FUNCTION_BLOCK SludgeBufferLogic_2 (* Composite Function Block Type *)
  (* Standard: 61499-2 *)
  (* Version 1.3, 10/1/2026, Claude/Hidryco, Schneider Electric, Rev1.3 - Revertidas as ligacoes de emergencia da Rev1.2 (FB_* e comando nos Av) que fechavam laco de eventos com a receita de emergencia; igual a Rev1.1 *)
  PACKAGE SE.Nereda;
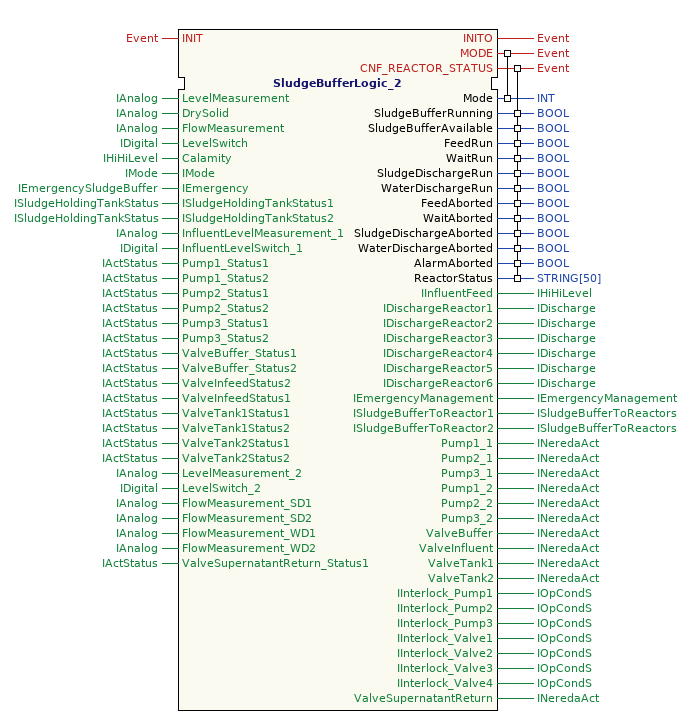
  EVENT_INPUT
    INIT; (* Initialization Request *)
  END_EVENT
  EVENT_OUTPUT
    INITO; (* Initialization Confirm *)
    MODE WITH Mode; (* Response from Socket *)
    CNF_REACTOR_STATUS WITH SludgeBufferRunning, SludgeBufferAvailable, FeedAborted, WaitAborted, SludgeDischargeAborted, WaterDischargeAborted, FeedRun, WaitRun, SludgeDischargeRun, WaterDischargeRun, AlarmAborted, ReactorStatus; (* Execution Confirmation *)
  END_EVENT
  VAR_OUTPUT
    Mode : INT; (* Response Data from Socket *)
    SludgeBufferRunning : BOOL; (* Result: IN1 OR IN2 OR ... *)
    SludgeBufferAvailable : BOOL; (* Result: IN1 AND IN2 AND ... *)
    FeedRun : BOOL;
    WaitRun : BOOL;
    SludgeDischargeRun : BOOL;
    WaterDischargeRun : BOOL;
    FeedAborted : BOOL;
    WaitAborted : BOOL;
    SludgeDischargeAborted : BOOL;
    WaterDischargeAborted : BOOL;
    AlarmAborted : BOOL; (* Result: IN1 OR IN2 OR ... *)
    ReactorStatus : STRING[50]; (* Output event qualifier *)
  END_VAR
  SOCKETS
    LevelMeasurement : IAnalog;
    DrySolid : IAnalog;
    FlowMeasurement : IAnalog;
    LevelSwitch : IDigital;
    Calamity : IHiHiLevel;
    IMode : IMode;
    IEmergency : IEmergencySludgeBuffer;
  END_SOCKETS
  SOCKETS
    ISludgeHoldingTankStatus1 : ISludgeHoldingTankStatus;
    ISludgeHoldingTankStatus2 : ISludgeHoldingTankStatus;
    InfluentLevelMeasurement_1 : IAnalog;
    InfluentLevelSwitch_1 : IDigital;
    Pump1_Status1 : IActStatus;
    Pump1_Status2 : IActStatus;
    Pump2_Status1 : IActStatus;
    Pump2_Status2 : IActStatus;
    Pump3_Status1 : IActStatus;
    Pump3_Status2 : IActStatus;
    ValveBuffer_Status1 : IActStatus;
    ValveBuffer_Status2 : IActStatus;
    ValveInfeedStatus2 : IActStatus;
    ValveInfeedStatus1 : IActStatus;
    ValveTank1Status1 : IActStatus;
    ValveTank1Status2 : IActStatus;
    ValveTank2Status1 : IActStatus;
    ValveTank2Status2 : IActStatus;
    LevelMeasurement_2 : IAnalog;
    LevelSwitch_2 : IDigital;
    FlowMeasurement_SD1 : IAnalog; (* 49FT0004 *)
    FlowMeasurement_SD2 : IAnalog; (* 49FT0004 *)
    FlowMeasurement_WD1 : IAnalog; (* 49FT0004 *)
    FlowMeasurement_WD2 : IAnalog; (* 49FT0004 *)
    ValveSupernatantReturn_Status1 : IActStatus; (* AV40001 status *)
  END_SOCKETS
  PLUGS
    IInfluentFeed : IHiHiLevel;
    IDischargeReactor1 : IDischarge;
    IDischargeReactor2 : IDischarge;
    IDischargeReactor3 : IDischarge;
    IDischargeReactor4 : IDischarge;
    IDischargeReactor5 : IDischarge;
    IDischargeReactor6 : IDischarge;
    IEmergencyManagement : IEmergencyManagement(pin_D997CA5474076632 := TRUE);
    ISludgeBufferToReactor1 : ISludgeBufferToReactors;
    ISludgeBufferToReactor2 : ISludgeBufferToReactors;
  END_PLUGS
  PLUGS
    Pump1_1 : INeredaAct;
    Pump2_1 : INeredaAct;
    Pump3_1 : INeredaAct;
    Pump1_2 : INeredaAct;
    Pump2_2 : INeredaAct;
    Pump3_2 : INeredaAct;
    ValveBuffer : INeredaAct;
    ValveInfluent : INeredaAct;
    ValveTank1 : INeredaAct;
    ValveTank2 : INeredaAct;
    IInterlock_Pump1 : IOpCondS; (* Condition summary chain output to downstream block *)
    IInterlock_Pump2 : IOpCondS;
    IInterlock_Pump3 : IOpCondS;
    IInterlock_Valve1 : IOpCondS; (* Condition summary chain output to downstream block *)
    IInterlock_Valve2 : IOpCondS;
    IInterlock_Valve3 : IOpCondS;
    IInterlock_Valve4 : IOpCondS;
    ValveSupernatantReturn : INeredaAct; (* AV40001 comando *)
  END_PLUGS
  (* 01 - FUNCTIONNAL INPUT INTERFACE *)
  (* 00 - INITIALIZATION *)
  (* 05 - LOGIC *)
  (* 06 - HMI INTERFACE *)
  (* 02 - FUNCTIONNAL OUTPUT INTERFACE *)
  (* Interlock *)
  (* 03 - FIELD INTERFACE *)
  (* Feed *)
  (* SludgeDischarge *)
  (* WaterDischarge *)
  (* Wait *)
  (* Check Phase Running / Check Phase Aborted *)
  FBS
    IThis : SludgeBufferLogic_2_HMI(QI := TRUE);
    LevelStatus : decodeStatus; {SET_ATTRIBUTE(Configuration.Component.HideUnusedPorts, )}
    Flow_Status : decodeStatus; {SET_ATTRIBUTE(Configuration.Component.HideUnusedPorts, )}
    LowLowBufferLevel : OR_88A3DD8EC65DD11C; {SET_ATTRIBUTE(Configuration.GenericFBType.InterfaceParams, Runtime.Standard#CNT:=2;OUT:BOOL)}
    LowLowLevel_pump1 : ilckCondItem(CondCause := Active1);
    HighHighCalamity : OR_88A3DD8EC65DD11C; {SET_ATTRIBUTE(Configuration.GenericFBType.InterfaceParams, Runtime.Standard#CNT:=2;OUT:BOOL)}
    HighHighLevel_Calamity_ValveBuffer : ilckCondItem(CondCause := Active1);
    DrySolidStatus : decodeStatus; {SET_ATTRIBUTE(Configuration.Component.HideUnusedPorts, )}
    LevelSwitchPv : INT2BOOL;
    HighHighLevel_Calamity_Pump1 : ilckCondItem(CondCause := Active1);
    HighHighLevel_Calamity_ValveInfeed : ilckCondItem(CondCause := Active1);
    HighHighLevel_Calamity_Pump2 : ilckCondItem(CondCause := Active1);
    HighHighLevel_Calamity_Pump3 : ilckCondItem(CondCause := Active1);
    HighHighLevel_Calamity_ValveTank2 : ilckCondItem(CondCause := Active1);
    LowLowLevel_pump2 : ilckCondItem(CondCause := Active1);
    LowLowLevel_pump3 : ilckCondItem(CondCause := Active1);
    HighHighLevel_Calamity_ValveTank1 : ilckCondItem(CondCause := Active1);
    FeedOCSLB2 : FeedOCSLB;
    Feed : Phase; {SET_ATTRIBUTE(Configuration.Component.HideUnusedPorts, )}
    SludgeDischargeOC : SludgeDischargeOCSLB;
    SludgeDischarge : Phase; {SET_ATTRIBUTE(Configuration.Component.HideUnusedPorts, )}
    WaterDischargeOC : WaterDischargeOCSLB;
    WaterDischarge : Phase; {SET_ATTRIBUTE(Configuration.Component.HideUnusedPorts, )}
    WaitOC : NoOC;
    Wait : Phase; {SET_ATTRIBUTE(Configuration.Component.HideUnusedPorts, )}
    CheckPhaseRunning : OR_169B00D031196E7C4; {SET_ATTRIBUTE(Configuration.GenericFBType.InterfaceParams, Runtime.Standard#CNT:=4;OUT:BOOL)}
    CheckPhaseAborted : OR_169B00D031196E7C4; {SET_ATTRIBUTE(Configuration.GenericFBType.InterfaceParams, Runtime.Standard#CNT:=4;OUT:BOOL)}
    SliudgeBufferAvalable : AND_169B00D031196E7C4; {SET_ATTRIBUTE(Configuration.GenericFBType.InterfaceParams, Runtime.Standard#CNT:=4;OUT:BOOL)}
    CheckPhaseInterlocked : OR_169B00D031196E7C4; {SET_ATTRIBUTE(Configuration.GenericFBType.InterfaceParams, Runtime.Standard#CNT:=4;OUT:BOOL)}
    FeedAv : CmdAndIlcked;
    WaitAv : CmdAndIlcked;
    CmdWait1 : NoCmd;
    CmdWait2 : NoCmd;
    SludgeDischargeAv : CmdAndIlcked;
    WaterDischargeAv : CmdAndIlcked;
    SludgeBufferStatus_21 : SludgeBufferStatus_2;
    CmdSludgeDischargeSLB1 : CmdSludgeDischargeSLB;
    CmdWaterDischargeSLB1 : CmdWaterDischargeSLB;
  END_FBS
  EVENT_CONNECTIONS
    LevelMeasurement.REQ_STATUS TO LevelStatus.REQ;
    FlowMeasurement.REQ_STATUS TO Flow_Status.REQ;
    LowLowBufferLevel.CNF TO LowLowLevel_pump1.REQ;
    CmdWaterDischargeSLB1.B72A275F8DEDE920 TO INITO;
    LevelStatus.CNF TO IDischargeReactor1.0F34BE432DD2288D;
    LevelStatus.CNF TO IDischargeReactor2.0F34BE432DD2288D;
    LevelStatus.CNF TO IInfluentFeed.15126F43E529BB4F;
    Calamity.15126F43E529BB4F TO HighHighCalamity.REQ;
    HighHighCalamity.CNF TO HighHighLevel_Calamity_ValveBuffer.REQ;
    DrySolid.REQ_STATUS TO DrySolidStatus.REQ;
    LevelSwitch.REQ TO LevelSwitchPv.DD5870AA881150BB;
    HighHighCalamity.CNF TO HighHighLevel_Calamity_Pump1.REQ;
    HighHighCalamity.CNF TO HighHighLevel_Calamity_Pump2.REQ;
    HighHighCalamity.CNF TO HighHighLevel_Calamity_Pump3.REQ;
    HighHighCalamity.CNF TO HighHighLevel_Calamity_ValveInfeed.REQ;
    HighHighCalamity.CNF TO HighHighLevel_Calamity_ValveTank2.REQ;
    LowLowBufferLevel.CNF TO LowLowLevel_pump2.REQ;
    LowLowBufferLevel.CNF TO LowLowLevel_pump3.REQ;
    HighHighCalamity.CNF TO HighHighLevel_Calamity_ValveTank1.REQ;
    IMode.MODE TO Feed.8CB9CCC96FA037F2;
    IMode.RESET TO Feed.0B9CBD1FB67738FF;
    IMode.MODE TO Wait.8CB9CCC96FA037F2;
    IMode.RESET TO Wait.0B9CBD1FB67738FF;
    IMode.MODE TO SludgeDischarge.8CB9CCC96FA037F2;
    IMode.RESET TO SludgeDischarge.0B9CBD1FB67738FF;
    IMode.MODE TO WaterDischarge.8CB9CCC96FA037F2;
    IMode.RESET TO WaterDischarge.0B9CBD1FB67738FF;
    IEmergencyManagement.33EC5B834E8FFAF3 TO IEmergencyManagement.12FB600C11F75EA2;
    CheckPhaseRunning.CNF TO CheckPhaseAborted.REQ;
    CheckPhaseAborted.CNF TO CheckPhaseInterlocked.REQ;
    Feed.C9D225E9FF976CF5 TO CheckPhaseRunning.REQ;
    Wait.C9D225E9FF976CF5 TO CheckPhaseRunning.REQ;
    WaterDischarge.C9D225E9FF976CF5 TO CheckPhaseRunning.REQ;
    WaterDischarge.C9D225E9FF976CF5 TO WaterDischargeAv.42EB462001E7FF11;
    SludgeDischarge.C9D225E9FF976CF5 TO SludgeDischargeAv.42EB462001E7FF11;
    Feed.C9D225E9FF976CF5 TO FeedAv.42EB462001E7FF11;
    Wait.C9D225E9FF976CF5 TO WaitAv.42EB462001E7FF11;
    SludgeDischarge.C9D225E9FF976CF5 TO CheckPhaseRunning.REQ;
    WaitAv.F9551E9B0D43115F TO SliudgeBufferAvalable.REQ;
    FeedAv.F9551E9B0D43115F TO SliudgeBufferAvalable.REQ;
    SludgeDischargeAv.F9551E9B0D43115F TO SliudgeBufferAvalable.REQ;
    WaterDischargeAv.F9551E9B0D43115F TO SliudgeBufferAvalable.REQ;
    IMode.MODE TO MODE;
    CheckPhaseAborted.CNF TO SludgeBufferStatus_21.2C4D36E78CFC061F;
    SludgeBufferStatus_21.B6E4C96ABAEB4E2A TO CNF_REACTOR_STATUS;
    IMode.MODE TO CmdSludgeDischargeSLB1.42062FCE2A6CF2D8;
    IMode.MODE TO CmdWaterDischargeSLB1.42062FCE2A6CF2D8;
    LevelStatus.CNF TO IDischargeReactor3.0F34BE432DD2288D;
    LevelStatus.CNF TO IDischargeReactor4.0F34BE432DD2288D;
    LevelStatus.CNF TO IDischargeReactor5.0F34BE432DD2288D;
    LevelStatus.CNF TO IDischargeReactor6.0F34BE432DD2288D;
    LevelSwitchPv.6FC99A5BD1C38561 TO IInfluentFeed.15126F43E529BB4F;
    WaterDischargeOC.C3BD2951F6A0C2EA TO CmdWaterDischargeSLB1.413C016DFFB59D18;
    CmdSludgeDischargeSLB1.B72A275F8DEDE920 TO WaterDischargeOC.EEE7655ECB3D19E4;
    SludgeDischargeOC.C3BD2951F6A0C2EA TO CmdSludgeDischargeSLB1.413C016DFFB59D18;
    WaitOC.C3BD2951F6A0C2EA TO CmdWait1.413C016DFFB59D18;
    CmdWait1.B72A275F8DEDE920 TO SludgeDischargeOC.EEE7655ECB3D19E4;
    CmdWait2.B72A275F8DEDE920 TO WaitOC.EEE7655ECB3D19E4;
    FeedOCSLB2.C3BD2951F6A0C2EA TO CmdWait2.413C016DFFB59D18;
    INIT TO IThis.73B62E902A5807A1;
    CmdWaterDischargeSLB1.B72A275F8DEDE920 TO IThis.559778F4ADF98A31;
    LevelMeasurement.REQ TO IThis.37C7911919BF6EA7;
    LevelStatus.CNF TO IThis.19121FA4406F1B6E;
    IThis.F68012C9A80C276B TO FeedOCSLB2.EEE7655ECB3D19E4;
    SliudgeBufferAvalable.CNF TO IEmergencyManagement.PHASE_NO_ABORTED;
    Feed.C9D225E9FF976CF5 TO ISludgeBufferToReactor1.C2C5F94C0FA89EA2;
    Feed.C9D225E9FF976CF5 TO ISludgeBufferToReactor2.C2C5F94C0FA89EA2;
    WaterDischarge.C9D225E9FF976CF5 TO Feed.58804E595E0ACE04;
    SludgeDischarge.C9D225E9FF976CF5 TO Feed.58804E595E0ACE04;
    Wait.C9D225E9FF976CF5 TO Feed.58804E595E0ACE04;
    IEmergency.37BB0210227B4D88 TO Feed.CC2F040586B1B15C;
    IEmergency.4D4A6D622AA6CDB1 TO Feed.4B853D9399632249;
    IEmergency.4D4A6D622AA6CDB1 TO Wait.4B853D9399632249;
    IEmergency.B8FB7A13CF18B1CA TO Wait.CC2F040586B1B15C;
    Feed.C9D225E9FF976CF5 TO Wait.58804E595E0ACE04;
    SludgeDischarge.C9D225E9FF976CF5 TO Wait.58804E595E0ACE04;
    WaterDischarge.C9D225E9FF976CF5 TO Wait.58804E595E0ACE04;
    Feed.C9D225E9FF976CF5 TO WaterDischarge.58804E595E0ACE04;
    Feed.C9D225E9FF976CF5 TO SludgeDischarge.58804E595E0ACE04;
    Wait.C9D225E9FF976CF5 TO SludgeDischarge.58804E595E0ACE04;
    IEmergency.7AF6A44EC4713EB1 TO SludgeDischarge.CC2F040586B1B15C;
    IEmergency.4D4A6D622AA6CDB1 TO SludgeDischarge.4B853D9399632249;
    IEmergency.6CE3EC6EFAA8A173 TO WaterDischarge.CC2F040586B1B15C;
    IEmergency.4D4A6D622AA6CDB1 TO WaterDischarge.4B853D9399632249;
    WaterDischarge.C9D225E9FF976CF5 TO SludgeDischarge.58804E595E0ACE04;
    SludgeDischarge.C9D225E9FF976CF5 TO WaterDischarge.58804E595E0ACE04;
    Wait.C9D225E9FF976CF5 TO WaterDischarge.58804E595E0ACE04;
    IEmergency.7AF6A44EC4713EB1 TO CmdSludgeDischargeSLB1.B960D5854AD6242C;
    IEmergency.6CE3EC6EFAA8A173 TO CmdWaterDischargeSLB1.B960D5854AD6242C;
    LevelStatus.CNF TO LowLowBufferLevel.REQ;
    LevelStatus.CNF TO CmdSludgeDischargeSLB1.AFC6599F2F80838F;
    LevelStatus.CNF TO CmdWaterDischargeSLB1.4D285A87325FFED2;
  END_CONNECTIONS
  DATA_CONNECTIONS
    LevelMeasurement.Status TO LevelStatus.Status;
    FlowMeasurement.Status TO Flow_Status.Status;
    LowLowBufferLevel.OUT TO LowLowLevel_pump1.CondSignal;
    LevelStatus.HiHiAlarm TO IInfluentFeed.C818324478A2F205;
    LevelStatus.HiHiAlarm TO IDischargeReactor1.F19118B95B2620C6;
    LevelStatus.HiHiAlarm TO IDischargeReactor2.F19118B95B2620C6;
    Calamity.C818324478A2F205 TO HighHighCalamity.IN1;
    Calamity.96B50ADF37756FFC TO HighHighCalamity.IN2;
    HighHighCalamity.OUT TO HighHighLevel_Calamity_ValveBuffer.CondSignal;
    DrySolid.Status TO DrySolidStatus.Status;
    LevelSwitch.Value TO LevelSwitchPv.4573FC8F228EB71D;
    HighHighCalamity.OUT TO HighHighLevel_Calamity_Pump1.CondSignal;
    HighHighCalamity.OUT TO HighHighLevel_Calamity_Pump2.CondSignal;
    HighHighCalamity.OUT TO HighHighLevel_Calamity_Pump3.CondSignal;
    HighHighCalamity.OUT TO HighHighLevel_Calamity_ValveInfeed.CondSignal;
    HighHighCalamity.OUT TO HighHighLevel_Calamity_ValveTank2.CondSignal;
    LevelStatus.LoAlarm TO LowLowBufferLevel.IN1;
    LowLowBufferLevel.OUT TO LowLowLevel_pump2.CondSignal;
    LowLowBufferLevel.OUT TO LowLowLevel_pump3.CondSignal;
    HighHighCalamity.OUT TO HighHighLevel_Calamity_ValveTank1.CondSignal;
    IMode.Mode TO Feed.60C668C3F76389FF;
    IMode.Reset TO Feed.3AA98D5129903FF7;
    IMode.Mode TO Wait.60C668C3F76389FF;
    IMode.Reset TO Wait.3AA98D5129903FF7;
    IMode.Mode TO SludgeDischarge.60C668C3F76389FF;
    IMode.Reset TO SludgeDischarge.3AA98D5129903FF7;
    IMode.Mode TO WaterDischarge.60C668C3F76389FF;
    IMode.Reset TO WaterDischarge.3AA98D5129903FF7;
    CheckPhaseRunning.OUT TO IEmergencyManagement.PhaseRun;
    CheckPhaseRunning.OUT TO SludgeBufferRunning;
    CheckPhaseAborted.OUT TO AlarmAborted;
    CheckPhaseAborted.OUT TO IEmergencyManagement.PhaseNoAborted;
    Feed.79A84BC5970E2DB6 TO CheckPhaseRunning.IN1;
    Wait.79A84BC5970E2DB6 TO CheckPhaseRunning.IN2;
    SludgeDischarge.79A84BC5970E2DB6 TO CheckPhaseRunning.IN3;
    WaterDischarge.79A84BC5970E2DB6 TO CheckPhaseRunning.IN4;
    Feed.9521593C56F0BC35 TO CheckPhaseAborted.IN1;
    Wait.9521593C56F0BC35 TO CheckPhaseAborted.IN2;
    SludgeDischarge.205C2090874C407F TO SludgeDischargeAv.FDADF7D226C9DBAE;
    Wait.205C2090874C407F TO WaitAv.FDADF7D226C9DBAE;
    Feed.205C2090874C407F TO FeedAv.FDADF7D226C9DBAE;
    WaterDischarge.205C2090874C407F TO WaterDischargeAv.FDADF7D226C9DBAE;
    SludgeDischarge.9521593C56F0BC35 TO CheckPhaseAborted.IN3;
    WaterDischarge.9521593C56F0BC35 TO CheckPhaseAborted.IN4;
    Feed.205C2090874C407F TO CheckPhaseInterlocked.IN1;
    Wait.205C2090874C407F TO CheckPhaseInterlocked.IN2;
    SludgeDischarge.205C2090874C407F TO CheckPhaseInterlocked.IN3;
    WaterDischarge.205C2090874C407F TO CheckPhaseInterlocked.IN4;
    FeedAv.11AB35620A02C8A5 TO SliudgeBufferAvalable.IN1;
    WaitAv.11AB35620A02C8A5 TO SliudgeBufferAvalable.IN2;
    SludgeDischargeAv.11AB35620A02C8A5 TO SliudgeBufferAvalable.IN3;
    WaterDischargeAv.11AB35620A02C8A5 TO SliudgeBufferAvalable.IN4;
    SliudgeBufferAvalable.OUT TO IEmergencyManagement.3C69BB1A066E9338;
    SliudgeBufferAvalable.OUT TO SludgeBufferAvailable;
    IMode.Mode TO Mode;
    Feed.79A84BC5970E2DB6 TO FeedRun;
    Wait.79A84BC5970E2DB6 TO WaitRun;
    SludgeDischarge.79A84BC5970E2DB6 TO SludgeDischargeRun;
    WaterDischarge.79A84BC5970E2DB6 TO WaterDischargeRun;
    Feed.9521593C56F0BC35 TO FeedAborted;
    Wait.9521593C56F0BC35 TO WaitAborted;
    SludgeDischarge.9521593C56F0BC35 TO SludgeDischargeAborted;
    WaterDischarge.9521593C56F0BC35 TO WaterDischargeAborted;
    CheckPhaseRunning.OUT TO SludgeBufferStatus_21.61016BEC47180831;
    CheckPhaseAborted.OUT TO SludgeBufferStatus_21.E9087AE335C18478;
    SludgeBufferStatus_21.407F4164D4F8FA5A TO ReactorStatus;
    IMode.Mode TO CmdSludgeDischargeSLB1.359E24E45FC44765;
    IMode.Mode TO CmdWaterDischargeSLB1.359E24E45FC44765;
    LevelStatus.HiHiAlarm TO IDischargeReactor3.F19118B95B2620C6;
    LevelStatus.HiHiAlarm TO IDischargeReactor4.F19118B95B2620C6;
    LevelStatus.HiHiAlarm TO IDischargeReactor6.F19118B95B2620C6;
    LevelStatus.HiHiAlarm TO IDischargeReactor5.F19118B95B2620C6;
    LevelSwitchPv.A6DEF5F9C27C1848 TO IInfluentFeed.96B50ADF37756FFC;
    LevelMeasurement.Value TO IThis.737770EE93C87B61;
    LevelMeasurement.ValueMin TO IThis.CABB298A467F63CE;
    LevelMeasurement.ValueMax TO IThis.5037DAC8B4AE8598;
    LevelStatus.HiHiAlarm TO IThis.91D28C0EF705C37F;
    Feed.9521593C56F0BC35 TO ISludgeBufferToReactor1.51FC34A07BFB4F2B;
    Feed.205C2090874C407F TO ISludgeBufferToReactor1.46E0963548A81AB0;
    Feed.9521593C56F0BC35 TO ISludgeBufferToReactor2.51FC34A07BFB4F2B;
    Feed.205C2090874C407F TO ISludgeBufferToReactor2.46E0963548A81AB0;
    Wait.D4263C4F5EA880F1 TO Feed.16DE804EA64A73FD;
    Wait.9521593C56F0BC35 TO Feed.8AE7594594AA7DBB;
    Wait.205C2090874C407F TO Feed.581756FA5F2310B2;
    SludgeDischarge.D4263C4F5EA880F1 TO Feed.B37A38F8606552EE;
    SludgeDischarge.9521593C56F0BC35 TO Feed.EFE2D0D8BEEEE5A1;
    SludgeDischarge.205C2090874C407F TO Feed.130A7AF73C88FF3B;
    WaterDischarge.D4263C4F5EA880F1 TO Feed.2E1C72C6FFE1DB32;
    WaterDischarge.9521593C56F0BC35 TO Feed.79BC17E07AAF4958;
    WaterDischarge.205C2090874C407F TO Feed.8FB896B12AF28D8B;
    IEmergency.0CCCE0E6A38C4CC4 TO Feed.195C6B3853E1CD26;
    IEmergency.A1711B52790021B0 TO Feed.2BB71ADCF214FB08;
    IEmergency.2D97C7DF176F1821 TO Wait.195C6B3853E1CD26;
    IEmergency.A1711B52790021B0 TO Wait.2BB71ADCF214FB08;
    Feed.D4263C4F5EA880F1 TO Wait.16DE804EA64A73FD;
    Feed.9521593C56F0BC35 TO Wait.8AE7594594AA7DBB;
    Feed.205C2090874C407F TO Wait.581756FA5F2310B2;
    SludgeDischarge.D4263C4F5EA880F1 TO Wait.B37A38F8606552EE;
    SludgeDischarge.9521593C56F0BC35 TO Wait.EFE2D0D8BEEEE5A1;
    SludgeDischarge.205C2090874C407F TO Wait.130A7AF73C88FF3B;
    WaterDischarge.D4263C4F5EA880F1 TO Wait.2E1C72C6FFE1DB32;
    WaterDischarge.9521593C56F0BC35 TO Wait.79BC17E07AAF4958;
    WaterDischarge.205C2090874C407F TO Wait.8FB896B12AF28D8B;
    Feed.D4263C4F5EA880F1 TO SludgeDischarge.16DE804EA64A73FD;
    Feed.9521593C56F0BC35 TO SludgeDischarge.8AE7594594AA7DBB;
    Feed.205C2090874C407F TO SludgeDischarge.581756FA5F2310B2;
    Feed.D4263C4F5EA880F1 TO WaterDischarge.16DE804EA64A73FD;
    Feed.9521593C56F0BC35 TO WaterDischarge.8AE7594594AA7DBB;
    Feed.205C2090874C407F TO WaterDischarge.581756FA5F2310B2;
    Wait.D4263C4F5EA880F1 TO SludgeDischarge.B37A38F8606552EE;
    Wait.9521593C56F0BC35 TO SludgeDischarge.EFE2D0D8BEEEE5A1;
    Wait.205C2090874C407F TO SludgeDischarge.130A7AF73C88FF3B;
    IEmergency.A1711B52790021B0 TO SludgeDischarge.2BB71ADCF214FB08;
    IEmergency.CC5E48971A6D3B85 TO SludgeDischarge.195C6B3853E1CD26;
    IEmergency.FDC6C047971AF4AB TO WaterDischarge.195C6B3853E1CD26;
    IEmergency.A1711B52790021B0 TO WaterDischarge.2BB71ADCF214FB08;
    WaterDischarge.D4263C4F5EA880F1 TO SludgeDischarge.2E1C72C6FFE1DB32;
    WaterDischarge.9521593C56F0BC35 TO SludgeDischarge.79BC17E07AAF4958;
    WaterDischarge.205C2090874C407F TO SludgeDischarge.8FB896B12AF28D8B;
    SludgeDischarge.D4263C4F5EA880F1 TO WaterDischarge.2E1C72C6FFE1DB32;
    SludgeDischarge.9521593C56F0BC35 TO WaterDischarge.79BC17E07AAF4958;
    SludgeDischarge.205C2090874C407F TO WaterDischarge.8FB896B12AF28D8B;
    Wait.D4263C4F5EA880F1 TO WaterDischarge.B37A38F8606552EE;
    Wait.9521593C56F0BC35 TO WaterDischarge.EFE2D0D8BEEEE5A1;
    Wait.205C2090874C407F TO WaterDischarge.130A7AF73C88FF3B;
    IEmergency.290CB544BD4AF7E0 TO CmdSludgeDischargeSLB1.6B6DC0CDC9D4BF59;
    IEmergency.D5F6310F45243454 TO CmdWaterDischargeSLB1.6B6DC0CDC9D4BF59;
    LevelStatus.LoAlarm TO CmdSludgeDischargeSLB1.261D74C13EDFD621;
    LevelStatus.LoAlarm TO CmdWaterDischargeSLB1.EB4DFF33F4044630;
  END_CONNECTIONS
  ADAPTER_CONNECTIONS
    HighHighLevel_Calamity_ValveTank2.ICondChainOut TO IInterlock_Valve3;
    HighHighLevel_Calamity_ValveInfeed.ICondChainOut TO IInterlock_Valve2;
    HighHighLevel_Calamity_ValveBuffer.ICondChainOut TO IInterlock_Valve1;
    HighHighLevel_Calamity_Pump1.ICondChainOut TO IInterlock_Pump1;
    HighHighLevel_Calamity_Pump2.ICondChainOut TO IInterlock_Pump2;
    HighHighLevel_Calamity_Pump3.ICondChainOut TO IInterlock_Pump3;
    LowLowLevel_pump1.ICondChainOut TO HighHighLevel_Calamity_Pump1.ICondChainIn;
    LowLowLevel_pump2.ICondChainOut TO HighHighLevel_Calamity_Pump2.ICondChainIn;
    LowLowLevel_pump3.ICondChainOut TO HighHighLevel_Calamity_Pump3.ICondChainIn;
    HighHighLevel_Calamity_ValveTank1.ICondChainOut TO IInterlock_Valve4;
    FeedOCSLB2.6B4386AEC7382B88 TO Feed.D86321A6D374FA01;
    SludgeDischargeOC.6B4386AEC7382B88 TO SludgeDischarge.D86321A6D374FA01;
    WaterDischargeOC.6B4386AEC7382B88 TO WaterDischarge.D86321A6D374FA01;
    WaitOC.6B4386AEC7382B88 TO Wait.D86321A6D374FA01;
    Feed.84E547B453517565 TO CmdWait2.E1021AA83C1C4121;
    Wait.84E547B453517565 TO CmdWait1.E1021AA83C1C4121;
    SludgeDischarge.84E547B453517565 TO CmdSludgeDischargeSLB1.E1021AA83C1C4121;
    CmdSludgeDischargeSLB1.73C2810D849D4A74 TO Pump2_1;
    CmdSludgeDischargeSLB1.11B726C8094295E9 TO Pump3_1;
    CmdSludgeDischargeSLB1.D7089B5E98615F78 TO ValveTank1;
    CmdSludgeDischargeSLB1.7AD0808434312B30 TO ValveTank2;
    WaterDischarge.84E547B453517565 TO CmdWaterDischargeSLB1.E1021AA83C1C4121;
    CmdWaterDischargeSLB1.F6607996697568B1 TO Pump1_2;
    CmdWaterDischargeSLB1.73C2810D849D4A74 TO Pump2_2;
    CmdWaterDischargeSLB1.11B726C8094295E9 TO Pump3_2;
    CmdWaterDischargeSLB1.D7089B5E98615F78 TO ValveBuffer;
    CmdWaterDischargeSLB1.7AD0808434312B30 TO ValveInfluent;
    Pump1_Status1 TO SludgeDischargeOC.426CA849096AFCF7;
    Pump2_Status1 TO SludgeDischargeOC.2B95FAAE91067885;
    Pump3_Status1 TO SludgeDischargeOC.FE2B4EB554D5332B;
    ValveTank1Status1 TO SludgeDischargeOC.AEF88E27D1E7B809;
    ValveTank2Status1 TO SludgeDischargeOC.B1059454EA1D3EB1;
    ValveBuffer_Status1 TO SludgeDischargeOC.E77AAE6AE2E77B57;
    ValveInfeedStatus1 TO SludgeDischargeOC.0FBECD124903C5D8;
    Pump1_Status2 TO WaterDischargeOC.8E8F96B83132E30C;
    Pump2_Status2 TO WaterDischargeOC.A28DD11F0C2A2D5D;
    Pump3_Status2 TO WaterDischargeOC.6F7C2D68D9E01EDF;
    ValveBuffer_Status2 TO WaterDischargeOC.DD370D907E1C7F85;
    ValveTank1Status2 TO WaterDischargeOC.EB6C0DCFCA843223;
    ValveTank2Status2 TO WaterDischargeOC.B8A0CBE6263B0FCB;
    InfluentLevelMeasurement_1 TO WaterDischargeOC.CCED8D64BDD673D1;
    InfluentLevelSwitch_1 TO WaterDischargeOC.3B098F5C14CCDC53;
    CmdSludgeDischargeSLB1.F6607996697568B1 TO Pump1_1;
    LevelMeasurement_2 TO FeedOCSLB2.48D5DE97F6AE4B6C;
    LevelSwitch_2 TO FeedOCSLB2.14B087BD2B49C1F0;
    ISludgeHoldingTankStatus1 TO SludgeDischargeOC.C3D97B62BC679D26;
    ISludgeHoldingTankStatus2 TO SludgeDischargeOC.F37E17D3A39C8811;
    ValveInfeedStatus2 TO WaterDischargeOC.D57E0E6283EBBD6E;
    FlowMeasurement_SD1 TO CmdSludgeDischargeSLB1.7E27CDF23DBBB407;
    FlowMeasurement_SD2 TO CmdSludgeDischargeSLB1.057735B6AA5D477A;
    FlowMeasurement_WD1 TO CmdWaterDischargeSLB1.7E27CDF23DBBB407;
    FlowMeasurement_WD2 TO CmdWaterDischargeSLB1.057735B6AA5D477A;
    CmdWaterDischargeSLB1.1B689F71B4B36D3B TO ValveSupernatantReturn;
    ValveSupernatantReturn_Status1 TO WaterDischargeOC.175174F4351C0854;
  END_CONNECTIONS
END_FUNCTION_BLOCK
